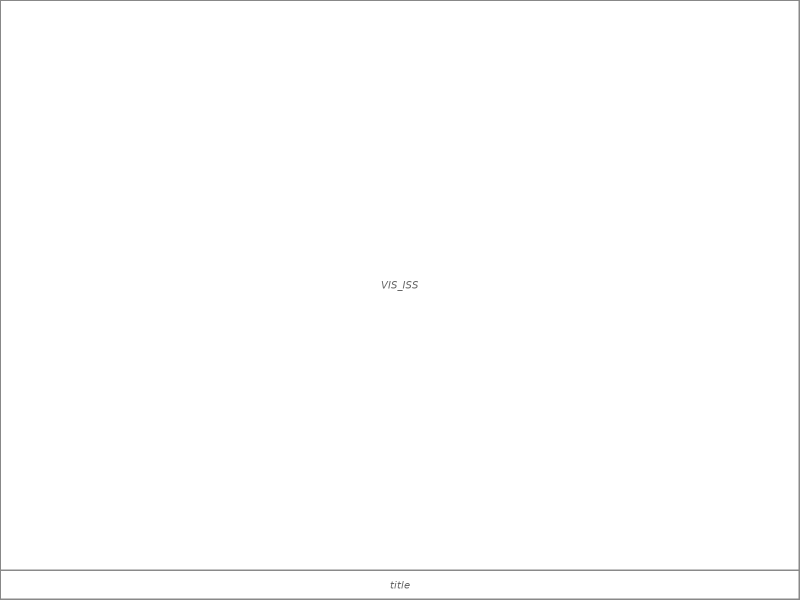
VISUALIZATION F5_InkSystem  // 800x600
    TabControl (0,0 800x570)
        shows VIS_ISS()
        shows VIS_MU()
        shows VIS_SpitUnit()
        shows VIS_Drip_purge()
        shows VIS_SubTank()
        [1]: TabTitle=MaintenanceUnit
        [2]: TabTitle=SpitUnit
        [3]: TabTitle=Drip_purge
        [4]: TabTitle=SubTank
    Frame (0,570 800x30)
        shows title()
END_VISUALIZATION

(* stored: Version 1.1.0.1, ProductVersion 3.1.4024.11
   Visu F5_InkSystem: Id {4cb0c248-19ab-4bf8-bfc7-9496d9939e63} *)
